FUNCTION "LAnyAxis_UnpubCamInMasterPosAxis" : Void
{ S7_Optimized_Access := 'TRUE' }
AUTHOR : 'tech.team.motioncontrol@siemens.com'
FAMILY : AnyAxis
VERSION : 1.0
   VAR_INPUT
      slave {InstructionName := 'TO_SynchronousAxis'; LibVersion := '5.0'} : TO_SynchronousAxis;
      master {InstructionName := 'TO_PositioningAxis'; LibVersion := '5.0'} : TO_PositioningAxis;
      cam {InstructionName := 'TO_Cam'; LibVersion := '5.0'} : TO_Cam;
   END_VAR

   VAR_IN_OUT
      instMC {InstructionName := 'MC_CAMIN'; LibVersion := '5.0'} : MC_CAMIN;
   END_VAR


BEGIN
	// Call of MC_Instruction
	#instMC(Master := #master,
	        Slave := #slave,
	        Cam := #cam);
END_FUNCTION

